PROGRAM MAIN
VAR
	fbMqttClient: FB_IotMqttClient; // MQTT client.       
    TopicToPublish   : STRING(255) := 'Temperatures'; // Mqtt topic on which we will broadcast the acual temperatures
    MessageToPublish : STRING(255); //String to send.
    fbSendMessageIntervalTimer : TON := (PT:=T#1S);	//Interval timer for broadcasting.
	ai_RoomTemperature AT %I* : INT; //Actual room temperature, linked to thermocouple	 
	
	TopicToPublishJson   : STRING(255) := 'unit1201/state'; //'homeassistant/sensor/unit_1400/config'; //'unit1201/state'; // Mqtt topic on which we will broadcast the acual temperatures in JSON format
	MessageToPublishJson : STRING(255); //String to send in JSON format
	mess				: STRING(1000) := '{"status":101}';
	//mess				: STRING ;
	fbJsonWriter : FB_JsonSaxWriter;
	fbJsonDataType : FB_JsonReadWriteDataType;
	TemperatureStructure:TemperatureStructure; 
	hadevice	:	HaDevice_1;	
	
	icount	:	INT;
	
	
	/// homeassistant/sensor/unit_1201/config
	
	(*
	{
  "name": "turned on",
  "state_topic": "unit1201/state",
  "unique_id": "unit_1201",
  "device": {
    "name": "smart enhed",
    "identifiers": [
      "unit_1201"
    ]
  }
}

"value_template": {% raw %}"{{ value_json.status }}"{% endraw %},
*)
	  


END_VAR

//mess := F_RTrim(mess1);

(*
hadevice.name			:= 'sensor2024';
hadevice.state_topic	:= 'unit1201/state';
hadevice.unique_id		:= 'unit_1400';
hadevice.value_template	:= '{{value_json.sensor2024 | round(2)}}';
hadevice.device.name	:= 'smart_enhed';
hadevice.device.identifiers[1]	:= 'smart_enhed';
hadevice.device.model			:= 'twincat3';
hadevice.device.manufacturer	:= 'beckhoff';
*)
IF _TaskInfo[GETCURTASKINDEXEX()].FirstCycle THEN    
    fbMqttClient.sHostName      := 'homeassistant'; // 192.168.2.159 - 100.97.177.128 - tailscale ip 100.92.234.119 - homeassistant
    fbMqttClient.nHostPort      := 1883;
	fbMqttClient.sUserName		:= 'twincat_xar';
	fbMqttClient.sUserPassword	:= '1234';
    fbMqttClient.sTopicPrefix   := '';     
	//fbMqttClient.sClientId 		:= 'Publishing PLC';
END_IF

fbMqttClient.Execute(TRUE);

IF fbMqttClient.bConnected THEN
    fbSendMessageIntervalTimer(IN:=TRUE);
    IF fbSendMessageIntervalTimer.Q THEN
        fbSendMessageIntervalTimer(IN:=FALSE);        
        MessageToPublish := CONCAT('Room temperature: ',REAL_TO_STRING(ai_RoomTemperature / 10.0));
		
        fbMqttClient.Publish(sTopic:= TopicToPublish, 
        	pPayload:= ADR(MessageToPublish), 
			nPayloadSize:= LEN2(ADR(MessageToPublish))+1, 
            eQoS:= TcIotMqttQos.AtMostOnceDelivery, 
			bRetain:= FALSE,
			bQueue:= FALSE);

			
			// Fill data
			IF hadevice.status <100 THEN
				hadevice.status := hadevice.status+1.11;
			END_IF
			IF hadevice.status > 20 THEN
			hadevice.status := 0;
			END_IF
			
			hadevice.sensor1 := 54;
			
			CASE icount OF
				0:
				IF hadevice.sensor2 <100 THEN
				hadevice.sensor2 := hadevice.sensor2+1;
				END_IF
				IF hadevice.sensor2 >= 20 THEN
					icount := 10;
				END_IF
				10:
				hadevice.sensor2 := hadevice.sensor2-1;
				IF hadevice.sensor2 <= 0 THEN
					icount := 0;
				END_IF
			END_CASE
			
		hadevice.sensor12 := 2024;	
	
			
			
			// COnvert to JSON string
			fbJsonWriter.ResetDocument();
			fbJsonDataType.AddJsonValueFromSymbol(fbJsonWriter, 'hadevice_1', SIZEOF(hadevice), ADR(hadevice));
			MessageToPublishJson := fbJsonWriter.GetDocument();
			fbJsonWriter.EndObject();
			fbJsonWriter.ResetDocument();
			
			//Publish
			fbMqttClient.Publish(sTopic:= TopicToPublishJson, 
        	pPayload:= ADR(MessageToPublishJson), 
			nPayloadSize:= LEN2(ADR(MessageToPublishJson)), 
            eQoS:= TcIotMqttQos.AtMostOnceDelivery, 
			bRetain:= FALSE,
			bQueue:= FALSE);
    END_IF
END_IF

TcIotMqttQos.AtLeastOnceDelivery;

END_PROGRAM

(* stored: Version 1.1.0.1, ProductVersion 3.1.4024.12
   POU MAIN: Id {0d666fc9-df30-40f9-b555-d1129e0440e1}, SpecialFunc None *)
